RoboDK station: Program_VDL_Testobject_AMR_mapped_example.rdk

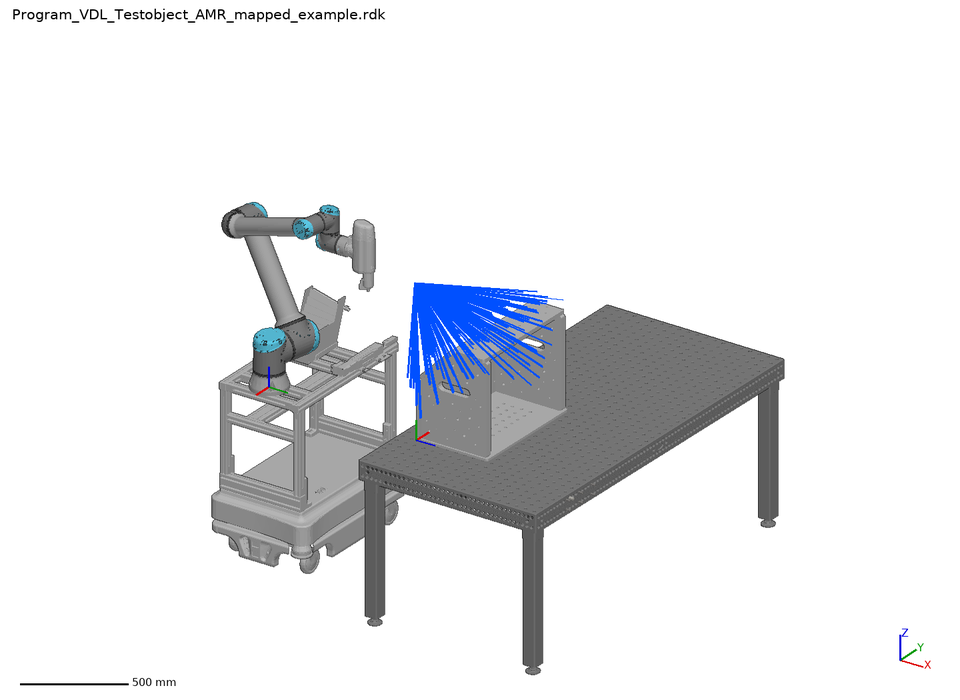
[picture v0: the station drawn from its stored meshes, robots at their saved joint values, targets as dots, program paths as lines]
Station Program_VDL_Testobject_AMR_mapped_example (saved by RoboDK 6.0.1). Poses are relative to the parent item; angles as X-Y-Z fixed-axis rotations.
Station parameters (name, value as stored): CollisionFreePlanner, UR10e, CollisionFreePlanner-Rob UR10e, Simplify-Mesh-Settings
  - object Lastafel at (0, 0, 0) mm, size 1021.8 x 2000 x 842 mm
  - object Lastafel_simplified at (0, 0, 0) mm, size 1000 x 2000 x 802.1 mm
  - frame UR10e Base at (-1716.15, 156.56, 116.62) mm, rotated rx 0 ry 0 rz -90 deg
    - robot UR10e: 6 axes, payload 10 kg, reach 1300 mm, repeatability 0.05 mm, weight 28.9 kg
        modified DH rows (alpha deg, a mm, theta deg, d mm): 0, 0, 0, 180.7; 90, 0, 180, 0; 0, 612.6, 0, 0; 0, 571.335, 0, 174.15; -90, 0, 0, 119.85; 90, 0, 180, 116.55
        joint limits [-180, -125, -30, -180, -180, -180] to [0, 0, 180, 180, 180, 180]; home [30.872, -95.296, 116.362, -22.187, 121.11, 179.827]; saved at [-101.47, -121.57, 102.82, 18.74, 78.53, -90]
      - tool schroevendraaier all in met nieuw kopstuk en tool, TCP at (210, -1, 100.6) mm, rotated rx 90 ry -90 rz 90 deg, size 86.2 x 139.7 x 345.9 mm, geometry from schroevendraaier all in met nieuw kopstuk en tool.STEP
      - tool tool simplified, TCP at (210, -1, 100.6) mm, rotated rx 90 ry -90 rz 90 deg, size 86.3 x 139.7 x 346 mm
    - object Assembly mir + frame aangepast naar ur10e versie 2 at (-733.08, 277.19, -552.66) mm, rotated rx 90 ry 0 rz 0.45 deg, size 901.1 x 1139.6 x 580.4 mm, geometry from Assembly mir + frame aangepast naar ur10e versie 2.STEP
    - object Mir + frame simplified at (-733.08, 277.19, -552.66) mm, rotated rx 90 ry 0 rz 0.45 deg, size 925.7 x 1139.7 x 582 mm
  - frame CSV Frame at (-919, 200, 49.99) mm, rotated rx 90 ry 0 rz 90.11 deg
    - object Test object at (0, 0.01, 0) mm, size 650 x 517 x 400 mm, geometry from Test object.STEP
    - object Test object simplified at (0, 0.01, 0) mm, size 650.1 x 517 x 436.5 mm
    - target pickup_m8 (joint target) at (672.95, 143.93, -450.44) mm, rotated rx 9.58 ry 86.75 rz -77.13 deg; joints [-45.747, -65.18, 99.078, -38.37, -45.221, -90.148] of UR10e
    - target Bovenpickup (joint target) at (657.59, 413.07, -465.55) mm, rotated rx 9.58 ry 86.75 rz -77.13 deg; joints [-45.787, -76.28, 85.202, -13.391, -45.26, -90.153] of UR10e
    - frame Type 1 at (0, 0, 0) mm
    - frame Type 2 at (0, 0, 0) mm
    - frame Type 3 at (0, 0, 0) mm
    - frame Type 4 at (0, 0, 0) mm
      - target Type 4_Instance 3 (joint target) at (23.3, 547, 301.7) mm, rotated rx 0 ry 90 rz -90 deg; joints [-102.885, -72.671, 92.625, 160.045, -77.004, 90.002, 10, 166.609] of UR10e
      - target Type 4_Instance 4 (joint target) at (23.3, 438.65, 75.94) mm, rotated rx 0 ry 45 rz -90 deg; joints [-103.104, -84.422, 87.706, -49.055, -99.303, -99.429, 10, 183.378] of UR10e
      - target Type 4_Instance 9 (joint target) at (26.7, 441.06, 78.35) mm, rotated rx 0 ry 45 rz -90 deg; joints [-102.796, -84.195, 87.209, -48.748, -99.088, -99.205, 10, 183.291] of UR10e
      - target Type 4_Instance 10 (joint target) at (26.7, 547, 298.3) mm, rotated rx 0 ry 90 rz -90 deg; joints [-102.681, -76.236, 72.773, 3.461, 77.208, -89.998, 10, 159.322] of UR10e
      - target Type 4_Instance 11 (joint target) at (23.3, 249.56, -30) mm, rotated rx 0 ry 0 rz -90 deg; joints [-113.843, -82.669, 125.473, 47.195, 89.998, 66.045, 10, 166.018] of UR10e
      - target Type 4_Instance 13 (joint target) at (626.7, 80.3, -30) mm, rotated rx 0 ry 0 rz -90 deg; joints [-47.849, -61.058, 119.335, -148.28, -90, -47.961, 10, 161.633] of UR10e
      - target Type 4_Instance 14 (joint target) at (626.7, 246.16, -30) mm, rotated rx 0 ry 0 rz -90 deg; joints [-47.849, -74.379, 115.27, -130.893, -90, -47.961, 10, 161.632] of UR10e
      - target Type 4_Instance 15 (joint target) at (623.3, 547, 301.7) mm, rotated rx 0 ry 90 rz -90 deg; joints [-60.97, -51.896, 61.186, 170.709, -118.918, 90.001, 10, 180] of UR10e
      - target Type 4_Instance 16 (joint target) at (623.3, 438.65, 75.94) mm, rotated rx 0 ry 45 rz -90 deg; joints [-60.972, -63.132, 60.541, -46.214, -70.007, -68.664, 10, 178.566] of UR10e
      - target Type 4_Instance 21 (joint target) at (626.7, 441.06, 78.35) mm, rotated rx 0 ry 45 rz -90 deg; joints [-60.862, -62.684, 59.637, -45.788, -69.934, -68.575, 10, 145.061] of UR10e
      - target Type 4_Instance 22 (joint target) at (626.7, 547, 298.3) mm, rotated rx 0 ry 90 rz -90 deg; joints [-60.689, -50.125, 33.926, 16.197, 119.199, -89.999, 10, 180] of UR10e
      - target Type 4_Instance 23 (joint target) at (623.3, 249.56, -30) mm, rotated rx 0 ry 0 rz -90 deg; joints [-48.052, -74.835, 115.447, -130.614, -90, -48.163, 10, 161.676] of UR10e
      - target Type 4_Instance 24 (joint target) at (623.3, 83.7, -30) mm, rotated rx 0 ry 0 rz -90 deg; joints [-48.052, -61.532, 119.625, -148.096, -90, -48.163, 10, 161.676] of UR10e
    - frame Type 5 at (0, 0, 0) mm
      - target Type 5_Instance 17 (joint target) at (690, 162.83, 229.27) mm, rotated rx 0 ry -90 rz 0 deg; joints [-46.016, -23.425, 44.903, -21.482, 133.871, 179.999, 10, 179.998] of UR10e
      - target Type 5_Instance 18 (joint target) at (690, 58.44, 67.81) mm, rotated rx 0 ry -90 rz 0 deg; joints [-39.55, -26.625, 63.718, -37.097, 140.338, 179.999, 10, 179.997] of UR10e
      - target Type 5_Instance 20 (joint target) at (690, 431.93, 203.64) mm, rotated rx 0 ry -90 rz 0 deg; joints [-45.071, -33.933, 37.797, -3.868, 134.816, 179.999, 10, 179.998] of UR10e
      - target Type 5_Instance 21 (joint target) at (690, 365.94, 282.45) mm, rotated rx 0 ry -90 rz 0 deg; joints [-47.885, -24.818, 26.79, -1.976, 132.002, 179.999, 10, 359.998] of UR10e
      - target Type 5_Instance 23 (joint target) at (690, 238.43, 67.81) mm, rotated rx 0 ry -90 rz 0 deg; joints [-39.549, -36.559, 63.061, -26.506, 140.338, 179.999, 10, 179.997] of UR10e
      - target Type 5_Instance 26 (joint target) at (690, 244.68, 61.56) mm, rotated rx 0 ry -90 rz 0 deg; joints [-39.274, -37.145, 63.508, -26.367, 140.613, 179.999, 10, 179.997] of UR10e
      - target Type 5_Instance 28 (joint target) at (690, 372.19, 276.2) mm, rotated rx 0 ry -90 rz 0 deg; joints [-47.672, -25.676, 27.854, -2.182, 132.215, 179.999, 10, 179.998] of UR10e
      - target Type 5_Instance 29 (joint target) at (690, 438.18, 197.39) mm, rotated rx 0 ry -90 rz 0 deg; joints [-44.836, -34.557, 38.349, -3.795, 135.051, 179.999, 10, 179.998] of UR10e
      - target Type 5_Instance 31 (joint target) at (690, 64.69, 61.56) mm, rotated rx 0 ry -90 rz 0 deg; joints [-39.274, -27.277, 64.367, -37.093, 140.613, 179.999, 10, 179.997] of UR10e
      - target Type 5_Instance 32 (joint target) at (690, 169.08, 223.02) mm, rotated rx 0 ry -90 rz 0 deg; joints [-45.788, -24.192, 45.805, -21.617, 134.099, 179.999, 10, 179.998] of UR10e
    - frame Type 6 at (0, 0, 0) mm
      - target Type 6_Instance 19 (joint target) at (690, 149.78, 155.18) mm, rotated rx 0 ry -90 rz 0 deg; joints [-43.202, -27.617, 54.989, -27.375, 136.685, 179.999, 10, 179.997] of UR10e
      - target Type 6_Instance 20 (joint target) at (690, 383.65, 150.69) mm, rotated rx 0 ry -90 rz 0 deg; joints [-43.024, -37.19, 48.814, -11.628, 136.864, 179.999, 10, 179.997] of UR10e
      - target Type 6_Instance 21 (joint target) at (690, 109.42, 53.94) mm, rotated rx 0 ry -90 rz 0 deg; joints [-38.935, -30.315, 65.385, -35.074, 140.952, 179.999, 10, 179.997] of UR10e
      - target Type 6_Instance 23 (joint target) at (690, 235, 198.1) mm, rotated rx 0 ry -90 rz 0 deg; joints [-44.863, -28.931, 48.337, -19.41, 135.024, 179.999, 10, 179.998] of UR10e
      - target Type 6_Instance 26 (joint target) at (690, 239.15, 193.95) mm, rotated rx 0 ry -90 rz 0 deg; joints [-44.706, -29.392, 48.814, -19.426, 135.181, 179.999, 10, 179.998] of UR10e
      - target Type 6_Instance 27 (joint target) at (690, 52.06, 164.48) mm, rotated rx 0 ry -90 rz 0 deg; joints [-43.57, -21.516, 53.32, -31.808, 136.318, 179.999, 10, 179.997] of UR10e
      - target Type 6_Instance 28 (joint target) at (690, 113.57, 49.79) mm, rotated rx 0 ry -90 rz 0 deg; joints [-38.749, -30.732, 65.764, -35.036, 141.138, 179.999, 10, 179.997] of UR10e
      - target Type 6_Instance 29 (joint target) at (690, 387.8, 146.54) mm, rotated rx 0 ry -90 rz 0 deg; joints [-42.857, -37.576, 49.111, -11.539, 137.03, 179.999, 10, 179.997] of UR10e
      - target Type 6_Instance 30 (joint target) at (690, 153.93, 151.03) mm, rotated rx 0 ry -90 rz 0 deg; joints [-43.037, -28.071, 55.459, -27.391, 136.85, 179.999, 10, 179.997] of UR10e
    - frame Type 7 at (0, 0, 0) mm
      - target Type 7_Instance 21 (joint target) at (690, 199.25, 90.33) mm, rotated rx 0 ry -90 rz 0 deg; joints [-40.527, -33.579, 61.56, -27.984, 139.36, 179.999, 10, 179.997] of UR10e
      - target Type 7_Instance 22 (joint target) at (690, 105.07, 210.14) mm, rotated rx 0 ry -90 rz 0 deg; joints [-45.314, -21.787, 47.822, -26.039, 134.573, 179.999, 10, 179.998] of UR10e
      - target Type 7_Instance 24 (joint target) at (690, 209.5, 240.26) mm, rotated rx 0 ry -90 rz 0 deg; joints [-46.413, -24.69, 42.513, -17.826, 133.475, 179.999, 10, 179.998] of UR10e
      - target Type 7_Instance 25 (joint target) at (690, 238.34, 130.69) mm, rotated rx 0 ry -90 rz 0 deg; joints [-42.216, -33.302, 56.657, -23.359, 137.671, 179.999, 10, 179.997] of UR10e
      - target Type 7_Instance 26 (joint target) at (690, 81.36, 108.27) mm, rotated rx 0 ry -90 rz 0 deg; joints [-41.288, -26.219, 60.011, -33.796, 138.6, 179.999, 10, 179.997] of UR10e
      - target Type 7_Instance 27 (joint target) at (690, 394.67, 226.16) mm, rotated rx 0 ry -90 rz 0 deg; joints [-45.903, -31.383, 36.687, -5.308, 133.984, 179.999, 10, 179.998] of UR10e
      - target Type 7_Instance 28 (joint target) at (690, 283.19, 75.59) mm, rotated rx 0 ry -90 rz 0 deg; joints [-39.89, -38.164, 61.229, -23.068, 139.997, 179.999, 10, 179.997] of UR10e
      - target Type 7_Instance 33 (joint target) at (690, 285.79, 72.99) mm, rotated rx 0 ry -90 rz 0 deg; joints [-39.777, -38.403, 61.402, -23.003, 140.11, 179.999, 10, 179.997] of UR10e
      - target Type 7_Instance 34 (joint target) at (690, 397.27, 223.56) mm, rotated rx 0 ry -90 rz 0 deg; joints [-45.808, -31.666, 36.968, -5.306, 134.079, 179.999, 10, 179.998] of UR10e
      - target Type 7_Instance 35 (joint target) at (690, 83.96, 105.67) mm, rotated rx 0 ry -90 rz 0 deg; joints [-41.178, -26.499, 60.301, -33.806, 138.709, 179.999, 10, 179.997] of UR10e
      - target Type 7_Instance 36 (joint target) at (690, 240.94, 128.09) mm, rotated rx 0 ry -90 rz 0 deg; joints [-42.11, -33.564, 56.89, -23.33, 137.778, 179.999, 10, 179.997] of UR10e
      - target Type 7_Instance 37 (joint target) at (690, 212.1, 237.66) mm, rotated rx 0 ry -90 rz 0 deg; joints [-46.319, -25.011, 42.886, -17.879, 133.568, 179.999, 10, 179.998] of UR10e
      - target Type 7_Instance 39 (joint target) at (690, 107.67, 207.54) mm, rotated rx 0 ry -90 rz 0 deg; joints [-45.217, -22.106, 48.206, -26.103, 134.67, 179.999, 10, 179.998] of UR10e
      - target Type 7_Instance 40 (joint target) at (690, 201.85, 87.73) mm, rotated rx 0 ry -90 rz 0 deg; joints [-40.415, -33.836, 61.78, -27.948, 139.472, 179.999, 10, 179.997] of UR10e
    - frame Type 8 at (0, 0, 0) mm
      - target Type 8_Instance 4 (joint target) at (690, 291.76, 278.38) mm, rotated rx 0 ry -90 rz 0 deg; joints [-47.747, -24.009, 32.664, -8.658, 132.14, 179.999, 10, 179.998] of UR10e
    - frame Type 9 at (0, 0, 0) mm
      - target Type 9_Instance 2 (joint target) at (690, 323.86, 128.14) mm, rotated rx 0 ry -90 rz 0 deg; joints [-42.112, -25.403, 57.919, 147.48, -137.776, -0.001, 10, 143.917] of UR10e
    - frame Type 10 at (0, 0, 0) mm
    - frame Type 11 at (0, 0, 0) mm
      - target Type 11_Instance 1 (joint target) at (-40, 496.62, 207.23) mm, rotated rx 0 ry 90 rz 0 deg; joints [-126.743, -62.581, 108.924, 133.657, -53.144, -179.998, 10, 131.763] of UR10e
      - target Type 11_Instance 3 (joint target) at (690, 496.62, 207.23) mm, rotated rx 0 ry -90 rz 0 deg; joints [-45.205, -29.153, 46.461, 162.688, -134.682, -0.001, 10, 147.532] of UR10e
    - frame Type 12 at (0, 0, 0) mm
      - target Type 12_Instance 1 (joint target) at (627.1, 245.76, -50) mm, rotated rx 0 ry 0 rz -90 deg; joints [-46.735, -75.219, 116.476, -131.259, -90, -46.846, 10, 161.058] of UR10e
      - target Type 12_Instance 2 (joint target) at (627.1, 79.9, -50) mm, rotated rx 0 ry 0 rz -90 deg; joints [-46.735, -61.643, 120.575, -148.934, -90, -46.847, 10, 161.059] of UR10e
      - target Type 12_Instance 4 (joint target) at (27.1, 245.76, -50) mm, rotated rx 0 ry 0 rz -90 deg; joints [-114.59, -84.24, 127.831, 46.409, 89.998, 65.298, 10, 165.308] of UR10e
      - target Type 12_Instance 5 (joint target) at (22.9, 249.96, -50) mm, rotated rx 0 ry 0 rz -90 deg; joints [-115.204, -84.589, 127.651, 46.938, 89.998, 64.684, 10, 164.952] of UR10e
      - target Type 12_Instance 7 (joint target) at (622.9, 84.1, -50) mm, rotated rx 0 ry 0 rz -90 deg; joints [-46.985, -62.238, 120.937, -148.701, -90, -47.097, 10, 161.109] of UR10e
      - target Type 12_Instance 8 (joint target) at (622.9, 249.96, -50) mm, rotated rx 0 ry 0 rz -90 deg; joints [-46.985, -75.793, 116.696, -130.905, -90, -47.096, 10, 161.109] of UR10e
      - target Type 12_Instance 9 (joint target) at (622.9, 452.51, 61.52) mm, rotated rx 0 ry 45 rz -90 deg; joints [-60.562, -64.309, 60.904, -45.513, -69.737, -68.335, 10, 173.428] of UR10e
      - target Type 12_Instance 10 (joint target) at (22.9, 452.51, 61.52) mm, rotated rx 0 ry 45 rz -90 deg; joints [-103.406, -67.579, 82.035, 119.739, 99.513, 80.353, 10, 176.518] of UR10e
      - target Type 12_Instance 11 (joint target) at (27.1, 455.48, 64.49) mm, rotated rx 0 ry 45 rz -90 deg; joints [-103.017, -67.369, 81.435, 120.174, 99.241, 80.635, 10, 176.628] of UR10e
      - target Type 12_Instance 12 (joint target) at (627.1, 455.48, 64.49) mm, rotated rx 0 ry 45 rz -90 deg; joints [-60.427, -63.751, 59.791, -44.996, -69.648, -68.226, 10, 178.598] of UR10e
      - target Type 12_Instance 13 (joint target) at (22.9, 567, 297.9) mm, rotated rx 0 ry 90 rz -90 deg; joints [-102.984, -73.629, 91.776, 161.852, -76.904, 90.002, 10, 167.651] of UR10e
      - target Type 12_Instance 14 (joint target) at (622.9, 567, 297.9) mm, rotated rx 0 ry 90 rz -90 deg; joints [-60.88, -49.539, 30.813, 18.725, 119.009, -89.999, 10, 180] of UR10e
      - target Type 12_Instance 15 (joint target) at (627.1, 567, 302.1) mm, rotated rx 0 ry 90 rz -90 deg; joints [-60.78, -51.911, 59.184, 172.726, -119.108, 90.001, 10, 180] of UR10e
      - target Type 12_Instance 16 (joint target) at (27.1, 567, 302.1) mm, rotated rx 0 ry 90 rz -90 deg; joints [-102.583, -75.695, 70.079, 5.615, 77.306, -89.998, 10, 158.65] of UR10e
    - frame Type 13 at (0, 0, 0) mm
      - target Type 13_Instance 1 (joint target) at (151.71, 262.13, -50) mm, rotated rx 0 ry 0 rz -90 deg; joints [-95.773, -83.432, 124.673, 48.758, 89.998, 84.115, 10, 174.113] of UR10e
      - target Type 13_Instance 2 (joint target) at (87.7, 197.43, -50) mm, rotated rx 0 ry 0 rz -90 deg; joints [-105.497, -79.491, 129.089, 40.401, 89.998, 74.391, 10, 9.724] of UR10e
      - target Type 13_Instance 3 (joint target) at (296.76, 181.09, -50) mm, rotated rx 0 ry 0 rz -90 deg; joints [-75.74, -71.409, 120.186, 41.221, 89.999, 104.148, 10, 29.757] of UR10e
      - target Type 13_Instance 4 (joint target) at (345.79, 276.43, -50) mm, rotated rx 0 ry 0 rz -90 deg; joints [-69.997, -75.802, 113.282, 52.519, 89.999, 109.892, 10, 11.297] of UR10e
      - target Type 13_Instance 5 (joint target) at (534.43, 161.34, -50) mm, rotated rx 0 ry 0 rz -90 deg; joints [-52.832, -57.756, 100.39, 47.364, 89.999, 127.057, 10, 18.046] of UR10e
      - target Type 13_Instance 6 (joint target) at (441.81, 52.38, -50) mm, rotated rx 0 ry 0 rz -90 deg; joints [-60.349, -54.367, 110.735, 33.63, 89.999, 119.539, 10, 13.734] of UR10e
      - target Type 13_Instance 7 (joint target) at (443.81, 54.38, -50) mm, rotated rx 0 ry 0 rz -90 deg; joints [-60.17, -54.448, 110.546, 33.9, 89.999, 119.719, 10, 0.27] of UR10e
      - target Type 13_Instance 8 (joint target) at (536.43, 163.34, -50) mm, rotated rx 0 ry 0 rz -90 deg; joints [-52.686, -57.769, 100.141, 47.626, 89.999, 127.202, 10, 13.726] of UR10e
      - target Type 13_Instance 9 (joint target) at (347.79, 278.43, -50) mm, rotated rx 0 ry 0 rz -90 deg; joints [-69.774, -75.816, 113.047, 52.767, 89.999, 110.114, 10, 18.047] of UR10e
      - target Type 13_Instance 10 (joint target) at (298.76, 183.09, -50) mm, rotated rx 0 ry 0 rz -90 deg; joints [-75.495, -71.483, 119.994, 41.487, 89.999, 104.393, 10, 11.28] of UR10e
      - target Type 13_Instance 11 (joint target) at (89.7, 199.43, -50) mm, rotated rx 0 ry 0 rz -90 deg; joints [-105.192, -79.644, 128.978, 40.664, 89.998, 74.696, 10, 29.697] of UR10e
      - target Type 13_Instance 12 (joint target) at (153.71, 264.13, -50) mm, rotated rx 0 ry 0 rz -90 deg; joints [-95.474, -83.521, 124.51, 49.01, 89.998, 84.415, 10, 9.719] of UR10e
      - target Type 13_Instance 13 (joint target) at (89.06, 404.63, 13.64) mm, rotated rx 0 ry 45 rz -90 deg; joints [-98.704, -70.334, 91.014, 113.978, 96.221, 83.741, 10, 177.621] of UR10e
      - target Type 13_Instance 14 (joint target) at (254.54, 497.09, 106.09) mm, rotated rx 0 ry 45 rz -90 deg; joints [-85.236, -77.888, 74.131, -41.339, -86.712, -86.707, 10, 178.988] of UR10e
      - target Type 13_Instance 15 (joint target) at (395.5, 427.75, 36.75) mm, rotated rx 0 ry 45 rz -90 deg; joints [-74.108, -78.948, 82.528, -49.682, -78.912, -78.699, 10, 176.271] of UR10e
      - target Type 13_Instance 16 (joint target) at (543.96, 434.97, 43.98) mm, rotated rx 0 ry 45 rz -90 deg; joints [-64.54, -70.739, 71.568, -48.726, -72.378, -71.48, 10, 174.162] of UR10e
      - target Type 13_Instance 17 (joint target) at (533.75, 507.68, 116.69) mm, rotated rx 0 ry 45 rz -90 deg; joints [-67.052, -64.398, 55.217, -38.156, -74.072, -73.418, 10, 178.849] of UR10e
      - target Type 13_Instance 18 (joint target) at (277.01, 427.75, 36.75) mm, rotated rx 0 ry 45 rz -90 deg; joints [-83.007, -83.56, 87.76, -49.408, -85.139, -85.122, 10, 181.559] of UR10e
      - target Type 13_Instance 19 (joint target) at (102, 474.94, 83.94) mm, rotated rx 0 ry 45 rz -90 deg; joints [-96.845, -83.195, 82.614, -44.632, -94.912, -94.931, 10, 181.766] of UR10e
      - target Type 13_Instance 20 (joint target) at (428.19, 391.63, 0.64) mm, rotated rx 0 ry 45 rz -90 deg; joints [-70.97, -80.099, 87.619, -54.112, -76.746, -76.376, 10, 175.4] of UR10e
      - target Type 13_Instance 21 (joint target) at (423.42, 466.27, 75.28) mm, rotated rx 0 ry 45 rz -90 deg; joints [-72.963, -74.418, 73.04, -44.891, -78.12, -77.856, 10, 176.142] of UR10e
      - target Type 13_Instance 22 (joint target) at (196.65, 410.41, 19.42) mm, rotated rx 0 ry 45 rz -90 deg; joints [-89.46, -87.308, 93.544, -51.238, -89.697, -89.697, 10, 179.428] of UR10e
      - target Type 13_Instance 23 (joint target) at (198.65, 411.83, 20.83) mm, rotated rx 0 ry 45 rz -90 deg; joints [-89.293, -87.142, 93.227, -51.088, -89.579, -89.579, 10, 179.234] of UR10e
      - target Type 13_Instance 24 (joint target) at (425.42, 467.68, 76.69) mm, rotated rx 0 ry 45 rz -90 deg; joints [-72.859, -74.197, 72.614, -44.703, -78.048, -77.779, 10, 176.123] of UR10e
      - target Type 13_Instance 25 (joint target) at (430.19, 393.05, 2.05) mm, rotated rx 0 ry 45 rz -90 deg; joints [-70.862, -79.903, 87.246, -53.953, -76.672, -76.296, 10, 175.381] of UR10e
      - target Type 13_Instance 26 (joint target) at (104, 476.35, 85.36) mm, rotated rx 0 ry 45 rz -90 deg; joints [-96.676, -83.034, 82.289, -44.458, -94.793, -94.811, 10, 181.722] of UR10e
      - target Type 13_Instance 27 (joint target) at (279.01, 429.16, 38.17) mm, rotated rx 0 ry 45 rz -90 deg; joints [-82.863, -64.806, 80.535, 119.054, 85.038, 94.98, 10, 181.652] of UR10e
      - target Type 13_Instance 28 (joint target) at (535.75, 509.1, 118.1) mm, rotated rx 0 ry 45 rz -90 deg; joints [-66.972, -64.113, 54.656, -37.897, -74.017, -73.356, 10, 178.848] of UR10e
      - target Type 13_Instance 29 (joint target) at (545.96, 436.39, 45.39) mm, rotated rx 0 ry 45 rz -90 deg; joints [-64.46, -70.508, 71.117, -48.524, -72.325, -71.418, 10, 174.153] of UR10e
      - target Type 13_Instance 30 (joint target) at (397.5, 429.16, 38.17) mm, rotated rx 0 ry 45 rz -90 deg; joints [-73.994, -78.746, 82.145, -49.517, -78.834, -78.615, 10, 176.249] of UR10e
      - target Type 13_Instance 31 (joint target) at (256.54, 498.5, 107.51) mm, rotated rx 0 ry 45 rz -90 deg; joints [-85.099, -77.687, 73.742, -41.157, -86.615, -86.61, 10, 178.958] of UR10e
      - target Type 13_Instance 32 (joint target) at (91.06, 406.05, 15.05) mm, rotated rx 0 ry 45 rz -90 deg; joints [-98.513, -70.235, 90.728, 114.18, 96.086, 83.878, 10, 177.675] of UR10e
      - target Type 13_Instance 33 (joint target) at (177.59, 567, 341.35) mm, rotated rx 0 ry 90 rz -90 deg; joints [-90.77, -69.872, 62.396, 7.474, 89.119, -89.998, 10, 178.087] of UR10e
      - target Type 13_Instance 34 (joint target) at (150.35, 567, 289.59) mm, rotated rx 0 ry 90 rz -90 deg; joints [-92.992, -75.716, 70.105, 5.609, 86.897, -89.998, 10, 157.205] of UR10e
      - target Type 13_Instance 35 (joint target) at (352.6, 567, 354.29) mm, rotated rx 0 ry 90 rz -90 deg; joints [-78.51, -61.995, 75.254, 166.739, -101.378, 90.001, 10, 180] of UR10e
      - target Type 13_Instance 36 (joint target) at (402.31, 567, 267.12) mm, rotated rx 0 ry 90 rz -90 deg; joints [-73.651, -68.989, 61.178, 7.81, 106.238, -89.999, 10, 180] of UR10e
      - target Type 13_Instance 37 (joint target) at (539.19, 567, 312.75) mm, rotated rx 0 ry 90 rz -90 deg; joints [-65.966, -56.633, 66.897, 169.735, -113.922, 90.001, 10, 180] of UR10e
      - target Type 13_Instance 38 (joint target) at (86.01, 567, 312.75) mm, rotated rx 0 ry 90 rz -90 deg; joints [-97.864, -71.97, 89.564, 162.404, -82.024, 90.002, 10, 161.954] of UR10e
      - target Type 13_Instance 39 (joint target) at (88.01, 567, 314.75) mm, rotated rx 0 ry 90 rz -90 deg; joints [-97.688, -71.77, 89.295, 162.474, -82.2, 90.002, 10, 160.487] of UR10e
      - target Type 13_Instance 40 (joint target) at (541.19, 567, 314.75) mm, rotated rx 0 ry 90 rz -90 deg; joints [-65.902, -55.187, 40.322, 14.863, 113.987, -89.999, 10, 180] of UR10e
      - target Type 13_Instance 41 (joint target) at (404.31, 567, 269.12) mm, rotated rx 0 ry 90 rz -90 deg; joints [-73.552, -67.097, 82.784, 164.311, -106.337, 90.001, 10, 180] of UR10e
      - target Type 13_Instance 42 (joint target) at (354.6, 567, 356.29) mm, rotated rx 0 ry 90 rz -90 deg; joints [-78.404, -62.246, 51.411, 10.834, 101.484, -89.999, 10, 180] of UR10e
      - target Type 13_Instance 43 (joint target) at (152.35, 567, 291.59) mm, rotated rx 0 ry 90 rz -90 deg; joints [-92.825, -73.045, 91.003, 162.041, -87.064, 90.002, 10, 167.384] of UR10e
      - target Type 13_Instance 44 (joint target) at (179.59, 567, 343.35) mm, rotated rx 0 ry 90 rz -90 deg; joints [-90.621, -69.618, 62.047, 7.569, 89.268, -89.998, 10, 180] of UR10e
    - frame Type 14 at (0, 0, 0) mm
      - target Type 14_Instance 1 (joint target) at (106.01, 54.36, -50) mm, rotated rx 0 ry 0 rz -90 deg; joints [-102.703, -64.218, 131.615, 22.602, 89.998, 77.185, 10, 167.184] of UR10e
      - target Type 14_Instance 2 (joint target) at (222.46, 140.16, -50) mm, rotated rx 0 ry 0 rz -90 deg; joints [-85.498, -70.689, 125.715, 34.972, 89.998, 94.39, 10, 17.205] of UR10e
      - target Type 14_Instance 3 (joint target) at (244.26, 249.8, -50) mm, rotated rx 0 ry 0 rz -90 deg; joints [-82.511, -79.049, 120.986, 48.062, 89.999, 97.377, 10, 13.089] of UR10e
      - target Type 14_Instance 4 (joint target) at (485.33, 106.11, -50) mm, rotated rx 0 ry 0 rz -90 deg; joints [-56.619, -56.58, 106.224, 40.354, 89.999, 123.27, 10, 25.893] of UR10e
      - target Type 14_Instance 5 (joint target) at (380.45, 161.27, -50) mm, rotated rx 0 ry 0 rz -90 deg; joints [-66.276, -65.945, 114.507, 41.436, 89.999, 113.612, 10, 9.658] of UR10e
      - target Type 14_Instance 6 (joint target) at (575.9, 260.02, -50) mm, rotated rx 0 ry 0 rz -90 deg; joints [-49.946, -60.821, 93.09, 57.729, 90, 129.942, 10, 21.418] of UR10e
      - target Type 14_Instance 9 (joint target) at (579.4, 263.52, -50) mm, rotated rx 0 ry 0 rz -90 deg; joints [-49.715, -79.73, 120.021, -130.293, -90, -49.827, 10, 162.963] of UR10e
      - target Type 14_Instance 10 (joint target) at (383.95, 164.77, -50) mm, rotated rx 0 ry 0 rz -90 deg; joints [-65.916, -83.306, 139.339, -146.035, -89.999, -66.028, 10, 19.318] of UR10e
      - target Type 14_Instance 11 (joint target) at (488.83, 109.61, -50) mm, rotated rx 0 ry 0 rz -90 deg; joints [-56.334, -71.353, 132.628, -151.277, -89.999, -56.446, 10, 11.952] of UR10e
      - target Type 14_Instance 12 (joint target) at (247.76, 253.3, -50) mm, rotated rx 0 ry 0 rz -90 deg; joints [-82.041, -79.148, 120.642, 48.505, 89.999, 97.848, 10, 199.782] of UR10e
      - target Type 14_Instance 13 (joint target) at (225.96, 143.66, -50) mm, rotated rx 0 ry 0 rz -90 deg; joints [-85.012, -70.901, 125.449, 35.451, 89.999, 94.877, 10, 13.053] of UR10e
      - target Type 14_Instance 14 (joint target) at (109.51, 57.86, -50) mm, rotated rx 0 ry 0 rz -90 deg; joints [-102.169, -64.579, 131.504, 23.075, 89.998, 77.719, 10, 17.157] of UR10e
      - target Type 14_Instance 15 (joint target) at (127.12, 439.74, 48.74) mm, rotated rx 0 ry 45 rz -90 deg; joints [-95.137, -67.739, 83.695, 118.922, 93.708, 86.283, 10, 178.61] of UR10e
      - target Type 14_Instance 16 (joint target) at (75.37, 511, 120.01) mm, rotated rx 0 ry 45 rz -90 deg; joints [-98.496, -79.783, 75.055, -40.598, -96.074, -96.109, 10, 182.107] of UR10e
      - target Type 14_Instance 17 (joint target) at (323.93, 466.7, 75.71) mm, rotated rx 0 ry 45 rz -90 deg; joints [-79.901, -78.538, 78.024, -44.925, -82.955, -82.902, 10, 177.714] of UR10e
      - target Type 14_Instance 18 (joint target) at (338.91, 394.47, 3.48) mm, rotated rx 0 ry 45 rz -90 deg; joints [-77.711, -83.896, 91.557, -53.315, -81.421, -81.324, 10, 176.938] of UR10e
      - target Type 14_Instance 19 (joint target) at (500.31, 456.11, 65.11) mm, rotated rx 0 ry 45 rz -90 deg; joints [-67.776, -71.43, 70.271, -46.028, -74.563, -73.97, 10, 174.963] of UR10e
      - target Type 14_Instance 20 (joint target) at (568.41, 403.62, 12.63) mm, rotated rx 0 ry 45 rz -90 deg; joints [-62.142, -71.633, 76.013, -52.872, -70.78, -69.596, 10, 173.468] of UR10e
      - target Type 14_Instance 21 (joint target) at (586.79, 502.82, 111.82) mm, rotated rx 0 ry 45 rz -90 deg; joints [-63.953, -61.535, 51.544, -38.046, -71.985, -71.022, 10, 178.751] of UR10e
      - target Type 14_Instance 22 (joint target) at (590.29, 505.29, 114.3) mm, rotated rx 0 ry 45 rz -90 deg; joints [-63.828, -60.998, 50.478, -37.547, -71.902, -70.924, 10, 178.751] of UR10e
      - target Type 14_Instance 23 (joint target) at (571.91, 406.1, 15.1) mm, rotated rx 0 ry 45 rz -90 deg; joints [-62.012, -71.249, 75.254, -52.531, -70.694, -69.493, 10, 173.455] of UR10e
      - target Type 14_Instance 24 (joint target) at (503.81, 458.58, 67.59) mm, rotated rx 0 ry 45 rz -90 deg; joints [-67.622, -71.022, 69.479, -45.675, -74.458, -73.853, 10, 174.941] of UR10e
      - target Type 14_Instance 25 (joint target) at (342.41, 396.95, 5.95) mm, rotated rx 0 ry 45 rz -90 deg; joints [-77.48, -83.571, 90.947, -53.055, -81.26, -81.157, 10, 177.844] of UR10e
      - target Type 14_Instance 26 (joint target) at (327.43, 469.18, 78.18) mm, rotated rx 0 ry 45 rz -90 deg; joints [-79.68, -78.182, 77.346, -44.622, -82.8, -82.743, 10, 177.669] of UR10e
      - target Type 14_Instance 27 (joint target) at (78.87, 513.48, 122.48) mm, rotated rx 0 ry 45 rz -90 deg; joints [-98.209, -79.489, 74.451, -40.267, -95.873, -95.904, 10, 182.034] of UR10e
      - target Type 14_Instance 28 (joint target) at (130.62, 442.21, 51.22) mm, rotated rx 0 ry 45 rz -90 deg; joints [-94.833, -67.524, 83.134, 119.282, 93.493, 86.499, 10, 178.691] of UR10e
      - target Type 14_Instance 29 (joint target) at (191.14, 567, 277.95) mm, rotated rx 0 ry 90 rz -90 deg; joints [-89.763, -73.515, 91.626, 161.888, -90.126, 90.002, 10, 169.322] of UR10e
      - target Type 14_Instance 30 (joint target) at (82.18, 567, 341.28) mm, rotated rx 0 ry 90 rz -90 deg; joints [-97.851, -71.351, 64.406, 6.944, 82.037, -89.998, 10, 180] of UR10e
      - target Type 14_Instance 31 (joint target) at (389.31, 567, 306.55) mm, rotated rx 0 ry 90 rz -90 deg; joints [-75.298, -64.65, 79.226, 165.422, -104.59, 90.001, 10, 180] of UR10e
      - target Type 14_Instance 32 (joint target) at (575.9, 567, 260.92) mm, rotated rx 0 ry 90 rz -90 deg; joints [-62.386, -58.227, 45.206, 13.02, 117.502, -89.999, 10, 180] of UR10e
      - target Type 14_Instance 33 (joint target) at (477.83, 567, 335.15) mm, rotated rx 0 ry 90 rz -90 deg; joints [-70.162, -58.097, 69.222, 168.874, -109.726, 90.001, 10, 180] of UR10e
      - target Type 14_Instance 34 (joint target) at (481.33, 567, 338.65) mm, rotated rx 0 ry 90 rz -90 deg; joints [-70.026, -56.918, 43.124, 13.793, 109.862, -89.999, 10, 180] of UR10e
      - target Type 14_Instance 35 (joint target) at (579.4, 567, 264.42) mm, rotated rx 0 ry 90 rz -90 deg; joints [-62.29, -58.108, 69.239, 168.867, -117.599, 90.001, 10, 180] of UR10e
      - target Type 14_Instance 36 (joint target) at (392.81, 567, 310.05) mm, rotated rx 0 ry 90 rz -90 deg; joints [-75.123, -65.264, 55.883, 9.38, 104.765, -89.999, 10, 180] of UR10e
      - target Type 14_Instance 37 (joint target) at (85.68, 567, 344.78) mm, rotated rx 0 ry 90 rz -90 deg; joints [-97.556, -70.949, 63.864, 7.084, 82.332, -89.998, 10, 164.515] of UR10e
      - target Type 14_Instance 38 (joint target) at (194.64, 567, 281.45) mm, rotated rx 0 ry 90 rz -90 deg; joints [-89.485, -75.57, 69.921, 5.648, 90.403, -89.998, 10, 156.577] of UR10e
    - frame Type 15 at (0, 0, 0) mm
      - target Type 15_Instance 1 (joint target) at (51.9, 254.25, -50) mm, rotated rx 0 ry 0 rz -90 deg; joints [-110.915, -84.792, 127.295, 47.496, 89.998, 68.974, 10, 158.972] of UR10e
      - target Type 15_Instance 2 (joint target) at (527.91, 90.81, -50) mm, rotated rx 0 ry 0 rz -90 deg; joints [-53.31, -53.292, 102.185, 41.105, 89.999, 126.578, 10, 57.604] of UR10e
      - target Type 15_Instance 3 (joint target) at (507.48, 216.79, -50) mm, rotated rx 0 ry 0 rz -90 deg; joints [-54.857, -62.795, 101.623, 51.17, 89.999, 125.031, 10, 10.064] of UR10e
      - target Type 15_Instance 4 (joint target) at (241.89, 72.42, -50) mm, rotated rx 0 ry 0 rz -90 deg; joints [-82.83, -63.421, 125.671, 27.749, 89.999, 97.058, 10, 27.973] of UR10e
      - target Type 15_Instance 5 (joint target) at (179.24, 197.73, -50) mm, rotated rx 0 ry 0 rz -90 deg; joints [-91.686, -77.34, 126.183, 41.155, 89.998, 88.203, 10, 13.919] of UR10e
      - target Type 15_Instance 6 (joint target) at (348.81, 216.79, -50) mm, rotated rx 0 ry 0 rz -90 deg; joints [-69.662, -71.658, 115.377, 46.279, 89.999, 110.227, 10, 22.024] of UR10e
      - target Type 15_Instance 7 (joint target) at (367.88, 80.6, -50) mm, rotated rx 0 ry 0 rz -90 deg; joints [-67.594, -59.834, 116.846, 32.986, 89.999, 112.294, 10, 13.292] of UR10e
      - target Type 15_Instance 8 (joint target) at (73.69, 134.39, -50) mm, rotated rx 0 ry 0 rz -90 deg; joints [-107.627, -73.455, 131.174, 32.28, 89.998, 72.261, 10, 40.033] of UR10e
      - target Type 15_Instance 9 (joint target) at (447.55, 154.82, -50) mm, rotated rx 0 ry 0 rz -90 deg; joints [-59.836, -62.081, 108.907, 43.172, 89.999, 120.053, 10, 47.792] of UR10e
      - target Type 15_Instance 10 (joint target) at (447.55, 272.63, -50) mm, rotated rx 0 ry 0 rz -90 deg; joints [-59.836, -69.676, 105.204, 54.469, 89.999, 120.053, 10, 11.297] of UR10e
      - target Type 15_Instance 11 (joint target) at (453.05, 278.13, -50) mm, rotated rx 0 ry 0 rz -90 deg; joints [-59.35, -69.646, 104.486, 55.158, 89.999, 120.539, 10, 0.718] of UR10e
      - target Type 15_Instance 12 (joint target) at (453.05, 160.32, -50) mm, rotated rx 0 ry 0 rz -90 deg; joints [-59.35, -62.186, 108.287, 43.897, 89.999, 120.539, 10, 11.261] of UR10e
      - target Type 15_Instance 13 (joint target) at (79.19, 139.89, -50) mm, rotated rx 0 ry 0 rz -90 deg; joints [-106.792, -73.969, 130.952, 33.016, 89.998, 73.096, 10, 47.442] of UR10e
      - target Type 15_Instance 14 (joint target) at (373.38, 86.1, -50) mm, rotated rx 0 ry 0 rz -90 deg; joints [-67.013, -60.092, 116.352, 33.738, 89.999, 112.875, 10, 39.779] of UR10e
      - target Type 15_Instance 15 (joint target) at (354.31, 222.29, -50) mm, rotated rx 0 ry 0 rz -90 deg; joints [-69.057, -71.765, 114.775, 46.988, 89.999, 110.832, 10, 13.25] of UR10e
      - target Type 15_Instance 16 (joint target) at (184.74, 203.23, -50) mm, rotated rx 0 ry 0 rz -90 deg; joints [-90.881, -77.639, 125.755, 41.883, 89.998, 89.007, 10, 21.824] of UR10e
      - target Type 15_Instance 17 (joint target) at (247.39, 77.92, -50) mm, rotated rx 0 ry 0 rz -90 deg; joints [-82.089, -63.818, 125.298, 28.518, 89.999, 97.799, 10, 13.821] of UR10e
      - target Type 15_Instance 18 (joint target) at (512.98, 222.29, -50) mm, rotated rx 0 ry 0 rz -90 deg; joints [-54.434, -62.788, 100.908, 51.878, 89.999, 125.455, 10, 27.656] of UR10e
      - target Type 15_Instance 19 (joint target) at (533.41, 96.31, -50) mm, rotated rx 0 ry 0 rz -90 deg; joints [-52.906, -53.4, 101.564, 41.834, 89.999, 126.983, 10, 10.044] of UR10e
      - target Type 15_Instance 20 (joint target) at (57.4, 259.75, -50) mm, rotated rx 0 ry 0 rz -90 deg; joints [-110.089, -85.175, 126.982, 48.192, 89.998, 69.799, 10, 57.183] of UR10e
      - target Type 15_Instance 21 (joint target) at (207.16, 459.25, 68.26) mm, rotated rx 0 ry 45 rz -90 deg; joints [-88.666, -82.793, 83.702, -45.917, -89.135, -89.135, 10, 179.777] of UR10e
      - target Type 15_Instance 22 (joint target) at (423.04, 512.22, 121.23) mm, rotated rx 0 ry 45 rz -90 deg; joints [-73.874, -51.829, 51.601, 134.093, 78.75, 101.473, 10, 176.463] of UR10e
      - target Type 15_Instance 23 (joint target) at (487.05, 404.36, 13.37) mm, rotated rx 0 ry 45 rz -90 deg; joints [-67.262, -76.203, 81.684, -52.774, -74.214, -73.578, 10, 174.605] of UR10e
      - target Type 15_Instance 24 (joint target) at (306.59, 512.22, 121.23) mm, rotated rx 0 ry 45 rz -90 deg; joints [-81.651, -74.665, 68.592, -39.225, -84.185, -84.155, 10, 178.192] of UR10e
      - target Type 15_Instance 25 (joint target) at (160.86, 508.85, 117.86) mm, rotated rx 0 ry 45 rz -90 deg; joints [-92.157, -78.881, 74.145, -40.288, -91.603, -91.605, 10, 180.601] of UR10e
      - target Type 15_Instance 26 (joint target) at (156.77, 385.58, -5.41) mm, rotated rx 0 ry 45 rz -90 deg; joints [-92.95, -70.434, 93.258, 112.134, 92.164, 87.834, 10, 179.118] of UR10e
      - target Type 15_Instance 27 (joint target) at (273.22, 385.58, -5.41) mm, rotated rx 0 ry 45 rz -90 deg; joints [-82.898, -87.02, 95.784, -53.979, -85.063, -85.045, 10, 171.827] of UR10e
      - target Type 15_Instance 28 (joint target) at (586.47, 456.37, 65.37) mm, rotated rx 0 ry 45 rz -90 deg; joints [-62.683, -66.343, 63.374, -45.383, -71.139, -70.024, 10, 173.885] of UR10e
      - target Type 15_Instance 29 (joint target) at (591.97, 460.25, 69.26) mm, rotated rx 0 ry 45 rz -90 deg; joints [-62.488, -65.637, 61.975, -44.741, -71.009, -69.869, 10, 173.866] of UR10e
      - target Type 15_Instance 30 (joint target) at (278.72, 389.47, -1.53) mm, rotated rx 0 ry 45 rz -90 deg; joints [-82.482, -86.537, 94.882, -53.586, -84.77, -84.748, 10, 172.047] of UR10e
      - target Type 15_Instance 31 (joint target) at (162.27, 389.47, -1.53) mm, rotated rx 0 ry 45 rz -90 deg; joints [-92.448, -70.13, 92.415, 112.685, 91.809, 88.189, 10, 179.253] of UR10e
      - target Type 15_Instance 32 (joint target) at (166.36, 512.74, 121.75) mm, rotated rx 0 ry 45 rz -90 deg; joints [-91.74, -78.366, 73.128, -39.778, -91.309, -91.31, 10, 180.501] of UR10e
      - target Type 15_Instance 33 (joint target) at (312.09, 516.11, 125.12) mm, rotated rx 0 ry 45 rz -90 deg; joints [-81.31, -74.056, 67.416, -38.684, -83.945, -83.911, 10, 178.122] of UR10e
      - target Type 15_Instance 34 (joint target) at (492.55, 408.25, 17.25) mm, rotated rx 0 ry 45 rz -90 deg; joints [-67.009, -75.632, 80.579, -52.294, -74.042, -73.384, 10, 174.568] of UR10e
      - target Type 15_Instance 35 (joint target) at (428.54, 516.11, 125.12) mm, rotated rx 0 ry 45 rz -90 deg; joints [-73.596, -51.079, 49.953, 134.95, 78.558, 101.677, 10, 175.171] of UR10e
      - target Type 15_Instance 36 (joint target) at (212.66, 463.14, 72.15) mm, rotated rx 0 ry 45 rz -90 deg; joints [-88.245, -82.298, 82.749, -45.464, -88.838, -88.838, 10, 179.676] of UR10e
      - target Type 15_Instance 37 (joint target) at (69.6, 567, 280.35) mm, rotated rx 0 ry 90 rz -90 deg; joints [-99.557, -77.699, 72.58, 5.118, 80.332, -89.998, 10, 153.844] of UR10e
      - target Type 15_Instance 38 (joint target) at (258.92, 567, 328.7) mm, rotated rx 0 ry 90 rz -90 deg; joints [-84.775, -68.968, 61.149, 7.818, 95.114, -89.999, 10, 180] of UR10e
      - target Type 15_Instance 39 (joint target) at (485.01, 567, 276.26) mm, rotated rx 0 ry 90 rz -90 deg; joints [-68.334, -62.598, 76.167, 166.429, -111.554, 90.001, 10, 180] of UR10e
      - target Type 15_Instance 40 (joint target) at (564.68, 567, 328.7) mm, rotated rx 0 ry 90 rz -90 deg; joints [-64.925, -51.408, 34.024, 17.383, 114.964, -89.999, 10, 180] of UR10e
      - target Type 15_Instance 41 (joint target) at (289.56, 567, 280.35) mm, rotated rx 0 ry 90 rz -90 deg; joints [-82.096, -70.613, 87.719, 162.893, -97.792, 90.001, 10, 163.714] of UR10e
      - target Type 15_Instance 42 (joint target) at (295.06, 567, 285.85) mm, rotated rx 0 ry 90 rz -90 deg; joints [-81.74, -72.001, 65.277, 6.723, 98.148, -89.999, 10, 180] of UR10e
      - target Type 15_Instance 43 (joint target) at (570.18, 567, 334.2) mm, rotated rx 0 ry 90 rz -90 deg; joints [-64.761, -52.925, 60.866, 172.057, -115.127, 90.001, 10, 180] of UR10e
      - target Type 15_Instance 44 (joint target) at (490.51, 567, 281.76) mm, rotated rx 0 ry 90 rz -90 deg; joints [-68.124, -62.402, 51.646, 10.754, 111.764, -89.999, 10, 180] of UR10e
      - target Type 15_Instance 45 (joint target) at (264.42, 567, 334.2) mm, rotated rx 0 ry 90 rz -90 deg; joints [-84.414, -66.688, 82.197, 164.49, -95.474, 90.001, 10, 180] of UR10e
      - target Type 15_Instance 46 (joint target) at (75.1, 567, 285.85) mm, rotated rx 0 ry 90 rz -90 deg; joints [-99.041, -77.103, 71.844, 5.258, 80.847, -89.998, 10, 154.99] of UR10e
    - frame Type 16 at (0, 0, 0) mm
      - target Type 16_Instance 2 (joint target) at (643.54, 310.54, -50) mm, rotated rx 0 ry 0 rz -90 deg; joints [-45.779, -78.117, 112.073, -123.959, -90, -45.89, 10, 160.874] of UR10e
      - target Type 16_Instance 4 (joint target) at (1.46, 305.54, -50) mm, rotated rx 0 ry 0 rz -90 deg; joints [-118.287, -88.67, 124.828, 53.842, 89.998, 61.602, 10, 163.181] of UR10e
      - target Type 16_Instance 5 (joint target) at (1.46, 539, 148) mm, rotated rx 0 ry 45 rz -90 deg; joints [-103.451, -76.948, 68.851, -37.714, -99.544, -99.68, 10, 183.232] of UR10e
      - target Type 16_Instance 6 (joint target) at (648.54, 539, 148) mm, rotated rx 0 ry 45 rz -90 deg; joints [-61.694, -51.142, 31.087, -28.555, -70.483, -69.24, 10, 41.757] of UR10e
      - target Type 16_Instance 7 (joint target) at (648.54, 368.99, -22) mm, rotated rx 0 ry 45 rz -90 deg; joints [-56.415, -68.765, 75.857, -57.26, -67.045, -64.941, 10, 172.013] of UR10e
      - target Type 16_Instance 8 (joint target) at (1.46, 368.99, -22) mm, rotated rx 0 ry 45 rz -90 deg; joints [-107.136, -93.134, 103.745, -56.93, -102.101, -102.382, 10, 50.721] of UR10e
      - target Type 16_Instance 9 (joint target) at (1.46, 567, 226.46) mm, rotated rx 0 ry 90 rz -90 deg; joints [-99.834, -31.748, 22.94, -171.193, 99.945, 90.001, 10, 202.047] of UR10e
      - target Type 16_Instance 10 (joint target) at (1.46, 567, 373.54) mm, rotated rx 0 ry 90 rz -90 deg; joints [-103.254, -68.18, 60.048, 8.13, 76.634, -89.998, 10, 153.126] of UR10e
      - target Type 16_Instance 11 (joint target) at (648.54, 567, 226.46) mm, rotated rx 0 ry 90 rz -90 deg; joints [-57.228, -56.394, 66.514, 169.878, -122.66, 90.001, 10, 180] of UR10e
      - target Type 16_Instance 12 (joint target) at (648.54, 567, 373.54) mm, rotated rx 0 ry 90 rz -90 deg; joints [-61.684, -43.594, 44.858, 178.735, -118.205, 90.001, 10, 21.656] of UR10e
  - program CollisionFreeProg (401 instructions, listed below)
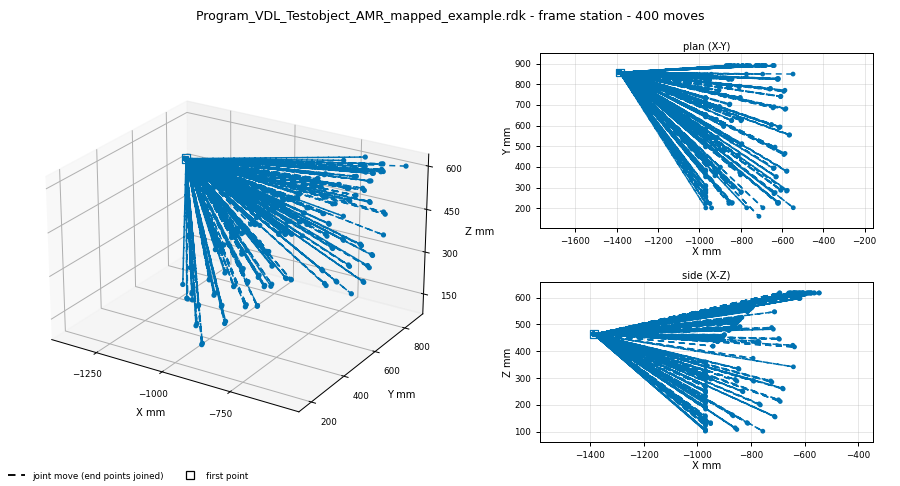
[picture p0: tool path of Program_VDL_Testobject_AMR_mapped_example.rdk in frame station, 400 of 400 moves have a stored position in this frame; points joined in program order, loops and branches not executed]

--- program CollisionFreeProg (robot UR10e) ---
  MoveJ (Bovenpickup)
  MoveJ (Type 4_Instance 3)
  MoveJ (Bovenpickup)
  MoveJ (Type 4_Instance 4)
  MoveJ (Bovenpickup)
  MoveJ (Type 4_Instance 9)
  MoveJ (Bovenpickup)
  MoveJ (Type 4_Instance 10)
  MoveJ (Bovenpickup)
  MoveJ (Type 4_Instance 11)
  MoveJ (Bovenpickup)
  MoveJ (Type 4_Instance 13)
  MoveJ (Bovenpickup)
  MoveJ (Type 4_Instance 14)
  MoveJ (Bovenpickup)
  MoveJ (Type 4_Instance 15)
  MoveJ (Bovenpickup)
  MoveJ (Type 4_Instance 16)
  MoveJ (Bovenpickup)
  MoveJ (Type 4_Instance 21)
  MoveJ (Bovenpickup)
  MoveJ (Type 4_Instance 22)
  MoveJ (Bovenpickup)
  MoveJ (Type 4_Instance 23)
  MoveJ (Bovenpickup)
  MoveJ (Type 4_Instance 24)
  MoveJ (Bovenpickup)
  MoveJ (Type 5_Instance 17)
  MoveJ (Bovenpickup)
  MoveJ (Type 5_Instance 18)
  MoveJ (Bovenpickup)
  MoveJ (Type 5_Instance 20)
  MoveJ (Bovenpickup)
  MoveJ (Type 5_Instance 21)
  MoveJ (Bovenpickup)
  MoveJ (Type 5_Instance 23)
  MoveJ (Bovenpickup)
  MoveJ (Type 5_Instance 26)
  MoveJ (Bovenpickup)
  MoveJ (Type 5_Instance 28)
  MoveJ (Bovenpickup)
  MoveJ (Type 5_Instance 29)
  MoveJ (Bovenpickup)
  MoveJ (Type 5_Instance 31)
  MoveJ (Bovenpickup)
  MoveJ (Type 5_Instance 32)
  MoveJ (Bovenpickup)
  MoveJ (Type 6_Instance 19)
  MoveJ (Bovenpickup)
  MoveJ (Type 6_Instance 20)
  MoveJ (Bovenpickup)
  MoveJ (Type 6_Instance 21)
  MoveJ (Bovenpickup)
  MoveJ (Type 6_Instance 23)
  MoveJ (Bovenpickup)
  MoveJ (Type 6_Instance 26)
  MoveJ (Bovenpickup)
  MoveJ (Type 6_Instance 27)
  MoveJ (Bovenpickup)
  MoveJ (Type 6_Instance 28)
  MoveJ (Bovenpickup)
  MoveJ (Type 6_Instance 29)
  MoveJ (Bovenpickup)
  MoveJ (Type 6_Instance 30)
  MoveJ (Bovenpickup)
  MoveJ (Type 7_Instance 21)
  MoveJ (Bovenpickup)
  MoveJ (Type 7_Instance 22)
  MoveJ (Bovenpickup)
  MoveJ (Type 7_Instance 24)
  MoveJ (Bovenpickup)
  MoveJ (Type 7_Instance 25)
  MoveJ (Bovenpickup)
  MoveJ (Type 7_Instance 26)
  MoveJ (Bovenpickup)
  MoveJ (Type 7_Instance 27)
  MoveJ (Bovenpickup)
  MoveJ (Type 7_Instance 28)
  MoveJ (Bovenpickup)
  MoveJ (Type 7_Instance 33)
  MoveJ (Bovenpickup)
  MoveJ (Type 7_Instance 34)
  MoveJ (Bovenpickup)
  MoveJ (Type 7_Instance 35)
  MoveJ (Bovenpickup)
  MoveJ (Type 7_Instance 36)
  MoveJ (Bovenpickup)
  MoveJ (Type 7_Instance 37)
  MoveJ (Bovenpickup)
  MoveJ (Type 7_Instance 39)
  MoveJ (Bovenpickup)
  MoveJ (Type 7_Instance 40)
  MoveJ (Bovenpickup)
  MoveJ (Type 8_Instance 4)
  MoveJ (Bovenpickup)
  MoveJ (Type 9_Instance 2)
  MoveJ (Bovenpickup)
  MoveJ (Type 11_Instance 1)
  MoveJ (Bovenpickup)
  MoveJ (Type 11_Instance 3)
  MoveJ (Bovenpickup)
  MoveJ (Type 12_Instance 1)
  MoveJ (Bovenpickup)
  MoveJ (Type 12_Instance 2)
  MoveJ (Bovenpickup)
  MoveJ (Type 12_Instance 4)
  MoveJ (Bovenpickup)
  MoveJ (Type 12_Instance 5)
  MoveJ (Bovenpickup)
  MoveJ (Type 12_Instance 7)
  MoveJ (Bovenpickup)
  MoveJ (Type 12_Instance 8)
  MoveJ (Bovenpickup)
  MoveJ (Type 12_Instance 9)
  MoveJ (Bovenpickup)
  MoveJ (Type 12_Instance 10)
  MoveJ (Bovenpickup)
  MoveJ (Type 12_Instance 11)
  MoveJ (Bovenpickup)
  MoveJ (Type 12_Instance 12)
  MoveJ (Bovenpickup)
  MoveJ (Type 12_Instance 13)
  MoveJ (Bovenpickup)
  MoveJ (Type 12_Instance 14)
  MoveJ (Bovenpickup)
  MoveJ (Type 12_Instance 15)
  MoveJ (Bovenpickup)
  MoveJ (Type 12_Instance 16)
  MoveJ (Bovenpickup)
  MoveJ (Type 13_Instance 1)
  MoveJ (Bovenpickup)
  MoveJ (Type 13_Instance 2)
  MoveJ (Bovenpickup)
  MoveJ (Type 13_Instance 3)
  MoveJ (Bovenpickup)
  MoveJ (Type 13_Instance 4)
  MoveJ (Bovenpickup)
  MoveJ (Type 13_Instance 5)
  MoveJ (Bovenpickup)
  MoveJ (Type 13_Instance 6)
  MoveJ (Bovenpickup)
  MoveJ (Type 13_Instance 7)
  MoveJ (Bovenpickup)
  MoveJ (Type 13_Instance 8)
  MoveJ (Bovenpickup)
  MoveJ (Type 13_Instance 9)
  MoveJ (Bovenpickup)
  MoveJ (Type 13_Instance 10)
  MoveJ (Bovenpickup)
  MoveJ (Type 13_Instance 11)
  MoveJ (Bovenpickup)
  MoveJ (Type 13_Instance 12)
  MoveJ (Bovenpickup)
  MoveJ (Type 13_Instance 13)
  MoveJ (Bovenpickup)
  MoveJ (Type 13_Instance 14)
  MoveJ (Bovenpickup)
  MoveJ (Type 13_Instance 15)
  MoveJ (Bovenpickup)
  MoveJ (Type 13_Instance 16)
  MoveJ (Bovenpickup)
  MoveJ (Type 13_Instance 17)
  MoveJ (Bovenpickup)
  MoveJ (Type 13_Instance 18)
  MoveJ (Bovenpickup)
  MoveJ (Type 13_Instance 19)
  MoveJ (Bovenpickup)
  MoveJ (Type 13_Instance 20)
  MoveJ (Bovenpickup)
  MoveJ (Type 13_Instance 21)
  MoveJ (Bovenpickup)
  MoveJ (Type 13_Instance 22)
  MoveJ (Bovenpickup)
  MoveJ (Type 13_Instance 23)
  MoveJ (Bovenpickup)
  MoveJ (Type 13_Instance 24)
  MoveJ (Bovenpickup)
  MoveJ (Type 13_Instance 25)
  MoveJ (Bovenpickup)
  MoveJ (Type 13_Instance 26)
  MoveJ (Bovenpickup)
  MoveJ (Type 13_Instance 27)
  MoveJ (Bovenpickup)
  MoveJ (Type 13_Instance 28)
  MoveJ (Bovenpickup)
  MoveJ (Type 13_Instance 29)
  MoveJ (Bovenpickup)
  MoveJ (Type 13_Instance 30)
  MoveJ (Bovenpickup)
  MoveJ (Type 13_Instance 31)
  MoveJ (Bovenpickup)
  MoveJ (Type 13_Instance 32)
  MoveJ (Bovenpickup)
  MoveJ (Type 13_Instance 33)
  MoveJ (Bovenpickup)
  MoveJ (Type 13_Instance 34)
  MoveJ (Bovenpickup)
  MoveJ (Type 13_Instance 35)
  MoveJ (Bovenpickup)
  MoveJ (Type 13_Instance 36)
  MoveJ (Bovenpickup)
  MoveJ (Type 13_Instance 37)
  MoveJ (Bovenpickup)
  MoveJ (Type 13_Instance 38)
  MoveJ (Bovenpickup)
  MoveJ (Type 13_Instance 39)
  MoveJ (Bovenpickup)
  MoveJ (Type 13_Instance 40)
  MoveJ (Bovenpickup)
  MoveJ (Type 13_Instance 41)
  MoveJ (Bovenpickup)
  MoveJ (Type 13_Instance 42)
  MoveJ (Bovenpickup)
  MoveJ (Type 13_Instance 43)
  MoveJ (Bovenpickup)
  MoveJ (Type 13_Instance 44)
  MoveJ (Bovenpickup)
  MoveJ (Type 14_Instance 1)
  MoveJ (Bovenpickup)
  MoveJ (Type 14_Instance 2)
  MoveJ (Bovenpickup)
  MoveJ (Type 14_Instance 3)
  MoveJ (Bovenpickup)
  MoveJ (Type 14_Instance 4)
  MoveJ (Bovenpickup)
  MoveJ (Type 14_Instance 5)
  MoveJ (Bovenpickup)
  MoveJ (Type 14_Instance 6)
  MoveJ (Bovenpickup)
  MoveJ (Type 14_Instance 9)
  MoveJ (Bovenpickup)
  MoveJ (Type 14_Instance 10)
  MoveJ (Bovenpickup)
  MoveJ (Type 14_Instance 11)
  MoveJ (Bovenpickup)
  MoveJ (Type 14_Instance 12)
  MoveJ (Bovenpickup)
  MoveJ (Type 14_Instance 13)
  MoveJ (Bovenpickup)
  MoveJ (Type 14_Instance 14)
  MoveJ (Bovenpickup)
  MoveJ (Type 14_Instance 15)
  MoveJ (Bovenpickup)
  MoveJ (Type 14_Instance 16)
  MoveJ (Bovenpickup)
  MoveJ (Type 14_Instance 17)
  MoveJ (Bovenpickup)
  MoveJ (Type 14_Instance 18)
  MoveJ (Bovenpickup)
  MoveJ (Type 14_Instance 19)
  MoveJ (Bovenpickup)
  MoveJ (Type 14_Instance 20)
  MoveJ (Bovenpickup)
  MoveJ (Type 14_Instance 21)
  MoveJ (Bovenpickup)
  MoveJ (Type 14_Instance 22)
  MoveJ (Bovenpickup)
  MoveJ (Type 14_Instance 23)
  MoveJ (Bovenpickup)
  MoveJ (Type 14_Instance 24)
  MoveJ (Bovenpickup)
  MoveJ (Type 14_Instance 25)
  MoveJ (Bovenpickup)
  MoveJ (Type 14_Instance 26)
  MoveJ (Bovenpickup)
  MoveJ (Type 14_Instance 27)
  MoveJ (Bovenpickup)
  MoveJ (Type 14_Instance 28)
  MoveJ (Bovenpickup)
  MoveJ (Type 14_Instance 29)
  MoveJ (Bovenpickup)
  MoveJ (Type 14_Instance 30)
  MoveJ (Bovenpickup)
  MoveJ (Type 14_Instance 31)
  MoveJ (Bovenpickup)
  MoveJ (Type 14_Instance 32)
  MoveJ (Bovenpickup)
  MoveJ (Type 14_Instance 33)
  MoveJ (Bovenpickup)
  MoveJ (Type 14_Instance 34)
  MoveJ (Bovenpickup)
  MoveJ (Type 14_Instance 35)
  MoveJ (Bovenpickup)
  MoveJ (Type 14_Instance 36)
  MoveJ (Bovenpickup)
  MoveJ (Type 14_Instance 37)
  MoveJ (Bovenpickup)
  MoveJ (Type 14_Instance 38)
  MoveJ (Bovenpickup)
  MoveJ (Type 15_Instance 1)
  MoveJ (Bovenpickup)
  MoveJ (Type 15_Instance 2)
  MoveJ (Bovenpickup)
  MoveJ (Type 15_Instance 3)
  MoveJ (Bovenpickup)
  MoveJ (Type 15_Instance 4)
  MoveJ (Bovenpickup)
  MoveJ (Type 15_Instance 5)
  MoveJ (Bovenpickup)
  MoveJ (Type 15_Instance 6)
  MoveJ (Bovenpickup)
  MoveJ (Type 15_Instance 7)
  MoveJ (Bovenpickup)
  MoveJ (Type 15_Instance 8)
  MoveJ (Bovenpickup)
  MoveJ (Type 15_Instance 9)
  MoveJ (Bovenpickup)
  MoveJ (Type 15_Instance 10)
  MoveJ (Bovenpickup)
  MoveJ (Type 15_Instance 11)
  MoveJ (Bovenpickup)
  MoveJ (Type 15_Instance 12)
  MoveJ (Bovenpickup)
  MoveJ (Type 15_Instance 13)
  MoveJ (Bovenpickup)
  MoveJ (Type 15_Instance 14)
  MoveJ (Bovenpickup)
  MoveJ (Type 15_Instance 15)
  MoveJ (Bovenpickup)
  MoveJ (Type 15_Instance 16)
  MoveJ (Bovenpickup)
  MoveJ (Type 15_Instance 17)
  MoveJ (Bovenpickup)
  MoveJ (Type 15_Instance 18)
  MoveJ (Bovenpickup)
  MoveJ (Type 15_Instance 19)
  MoveJ (Bovenpickup)
  MoveJ (Type 15_Instance 20)
  MoveJ (Bovenpickup)
  MoveJ (Type 15_Instance 21)
  MoveJ (Bovenpickup)
  MoveJ (Type 15_Instance 22)
  MoveJ (Bovenpickup)
  MoveJ (Type 15_Instance 23)
  MoveJ (Bovenpickup)
  MoveJ (Type 15_Instance 24)
  MoveJ (Bovenpickup)
  MoveJ (Type 15_Instance 25)
  MoveJ (Bovenpickup)
  MoveJ (Type 15_Instance 26)
  MoveJ (Bovenpickup)
  MoveJ (Type 15_Instance 27)
  MoveJ (Bovenpickup)
  MoveJ (Type 15_Instance 28)
  MoveJ (Bovenpickup)
  MoveJ (Type 15_Instance 29)
  MoveJ (Bovenpickup)
  MoveJ (Type 15_Instance 30)
  MoveJ (Bovenpickup)
  MoveJ (Type 15_Instance 31)
  MoveJ (Bovenpickup)
  MoveJ (Type 15_Instance 32)
  MoveJ (Bovenpickup)
  MoveJ (Type 15_Instance 33)
  MoveJ (Bovenpickup)
  MoveJ (Type 15_Instance 34)
  MoveJ (Bovenpickup)
  MoveJ (Type 15_Instance 35)
  MoveJ (Bovenpickup)
  MoveJ (Type 15_Instance 36)
  MoveJ (Bovenpickup)
  MoveJ (Type 15_Instance 37)
  MoveJ (Bovenpickup)
  MoveJ (Type 15_Instance 38)
  MoveJ (Bovenpickup)
  MoveJ (Type 15_Instance 39)
  MoveJ (Bovenpickup)
  MoveJ (Type 15_Instance 40)
  MoveJ (Bovenpickup)
  MoveJ (Type 15_Instance 41)
  MoveJ (Bovenpickup)
  MoveJ (Type 15_Instance 42)
  MoveJ (Bovenpickup)
  MoveJ (Type 15_Instance 43)
  MoveJ (Bovenpickup)
  MoveJ (Type 15_Instance 44)
  MoveJ (Bovenpickup)
  MoveJ (Type 15_Instance 45)
  MoveJ (Bovenpickup)
  MoveJ (Type 15_Instance 46)
  MoveJ (Bovenpickup)
  MoveJ (Type 16_Instance 2)
  MoveJ (Bovenpickup)
  MoveJ (Type 16_Instance 4)
  MoveJ (Bovenpickup)
  MoveJ (Type 16_Instance 5)
  MoveJ (Bovenpickup)
  MoveJ (Type 16_Instance 6)
  MoveJ (Bovenpickup)
  MoveJ (Type 16_Instance 7)
  MoveJ (Bovenpickup)
  MoveJ (Type 16_Instance 8)
  MoveJ (Bovenpickup)
  MoveJ (Type 16_Instance 9)
  MoveJ (Bovenpickup)
  MoveJ (Type 16_Instance 10)
  MoveJ (Bovenpickup)
  MoveJ (Type 16_Instance 11)
  MoveJ (Bovenpickup)
  MoveJ (Type 16_Instance 12)
  Set IO_5=1
